TYPE ST_CFG_MovableStopAddonEmulation :
(**************************************************************************************
 * 	Application		:	BoxControl Framework
 *	Revision		:	$Revision:  $
 *	Revision date	:	$Date:  $
 *	Last changed by	:	$Author: q8hedls $
 *	URL				:	$URL:  $
 *
 *	Purpose			:	Scanner emulation configuration
 *
 * ------------------------------------------------------------------------------------
 *	Copyright Swisslog [IP AG], Switzerland. All rights reserved.
 * 
 * ------------------------------------------------------------------------------------
 *	
 * 	Revision History: 
 *
 * 	VERSION			DATE			INITIALS			DESCRIPTION
 *	0.1				01.01.2001		swl					Example
 *
 **************************************************************************************)
STRUCT
	Position_Max_Down				: INT;
	Position_Max_Up	  				: INT;	
	Position_Down					: INT;
	Position_Up	  					: INT;
END_STRUCT
END_TYPE

(* stored: Version 1.1.0.1, ProductVersion 3.1.4024.9
   DUT ST_CFG_MovableStopAddonEmulation: Id {3fc64d36-e9a1-4e27-868c-3bf06fb40a07} *)
